(* IEC 61131-3 sources: std_i2980_v2.06_cp053/Source/IMM/ieccontrol/OutputCoordination1 (part 2) *)

(* ---- ABCoordList.pu ---- *)
IMPORT_OVER_LISTFILE
 SET_ALARM
, tsListStructCoord
, tsDeviceId
, FBDebugTrace
, tsTraceLevel
, tsElementCoord
, tsSearchDataCoord

END_IMPORT

ALGORITHM_BLOCK ABCoordList #DUMMY_EDIT_BLOCK

SYSTEM_VAR
 sv_DeviceId : tsDeviceId;
 sv_TraceLevel : tsTraceLevel;
END_VAR

SYSTEM_OBJECT
 erListOverflow : ALARM;
END_OBJECT

VAR
 mListStruct : tsListStructCoord;
 miNextFree : DINT;
 miLowBound : DINT;
 miHighBound : DINT;
 mbInit : BOOL;
 miLastFound : DINT;
 miActElement : DINT;
 fbDebugTrace : FBDebugTrace;
END_VAR

ALGORITHM aInit

#BEGIN_EDIT_BLOCK
miLowBound := GET_LOW_BOUND(mListStruct.List);
miHighBound := GET_HIGH_BOUND(mListStruct.List);
miNextFree := miLowBound;
miLastFound := miLowBound;
miActElement := miLowBound;
mbInit := TRUE;

;#END_EDIT_BLOCK END_ALGORITHM

ALGORITHM aAdd

VAR_INPUT
 Element : tsElementCoord;
END_VAR
#BEGIN_EDIT_BLOCK
IF NOT mbInit THEN RETURN;; END_IF;

IF miNextFree < miHighBound THEN

    mListStruct.List[miNextFree] := Element;
    mListStruct.Used[miNextFree] := TRUE;
    miNextFree := miNextFree + 1;
ELSE
    //error: List Full
    SET_ALARM(Name := erListOverflow,
              SubID1 := sv_DeviceId.CompId,
              SubID2 := sv_DeviceId.IndexId,
              Param1 := 'ABCoordList.aAdd');
END_IF;

;#END_EDIT_BLOCK END_ALGORITHM

ALGORITHM aAddAt

VAR_INPUT
 Element : tsElementCoord;
 iPos : DINT;
END_VAR

VAR_TEMP
 i : DINT;
END_VAR

VAR
 iStart : DINT;
 iEnd : DINT;
END_VAR
#BEGIN_EDIT_BLOCK
IF NOT mbInit THEN RETURN; END_IF;

IF miNextFree <= miHighBound THEN
    IF iPos < miHighBound AND iPos >= miLowBound THEN

        IF iPos < miNextFree THEN

            iStart := miNextFree;
            iEnd := iPos+1;
        ELSE
            i := iPos;
            iEnd := miNextFree;
        END_IF;
        miNextFree := i + 1;

        //reorganize list
        FOR i := iStart TO iEnd BY -1 DO
            mListStruct.List[i] := mListStruct.List[i-1];
            mListStruct.Used[i] := TRUE;
        END_FOR;
        //adding Element
        mListStruct.List[iPos] := Element;
        mListStruct.Used[iPos] := TRUE;
    ELSE
        //error: out of bounds
        IF sv_TraceLevel.bApplication THEN
            fbDebugTrace(sText := 'ABCoordList.aAddAt: Error: Out of ListBounds');
        END_IF;
    END_IF;
ELSE
    //error: List Full
    SET_ALARM(Name := erListOverflow,
            SubID1 := sv_DeviceId.CompId,
            SubID2 := sv_DeviceId.IndexId,
            Param1 := 'ABCoordList.aAddAt');
END_IF;

;#END_EDIT_BLOCK END_ALGORITHM

ALGORITHM aSearch

VAR_INPUT
 SearchData : tsSearchDataCoord;
END_VAR

VAR_OUTPUT
 Element : tsElementCoord;
 iPos : DINT;
 bFound : BOOL;
END_VAR

VAR_TEMP
 i : DINT;
END_VAR
#BEGIN_EDIT_BLOCK
IF NOT mbInit THEN RETURN; END_IF;

iPos := 0;
bFound := FALSE;

FOR i := miLowBound TO miNextFree-1 DO

    IF  mListStruct.Used[i] THEN
        IF mListStruct.List[i].SearchData = SearchData THEN

            Element := mListStruct.List[i];
            //remember foundposition for aSearchNext
            miLastFound := i;
            iPos := i;
            bFound := TRUE;
            RETURN;
        END_IF;
    ELSE
        EXIT;
    END_IF;
END_FOR;

;#END_EDIT_BLOCK END_ALGORITHM

ALGORITHM aSearchNext

VAR_INPUT
 SearchData : tsSearchDataCoord;
END_VAR

VAR_OUTPUT
 Element : tsElementCoord;
 iPos : DINT;
 bFound : BOOL;
END_VAR

VAR_TEMP
 i : DINT;
END_VAR
#BEGIN_EDIT_BLOCK
IF NOT mbInit THEN RETURN;; END_IF;

iPos := 0;
bFound := FALSE;

FOR i := miLastFound+1 TO miNextFree-1 DO

    IF mListStruct.List[i].SearchData = SearchData THEN

       Element := mListStruct.List[i];
       //remember foundposition for then next aSearchNext
       miLastFound := i;
       iPos := i;
       bFound := TRUE;
       RETURN;;
    END_IF;
END_FOR;

;#END_EDIT_BLOCK END_ALGORITHM

ALGORITHM aRemove

VAR_INPUT
 SearchData : tsSearchDataCoord;
END_VAR

VAR_OUTPUT
 Element : tsElementCoord;
 iPos : DINT;
 bFound : BOOL;
END_VAR

VAR_TEMP
 i : DINT;
END_VAR
#BEGIN_EDIT_BLOCK
IF NOT mbInit THEN RETURN; END_IF;

iPos := 0;
bFound := FALSE;

FOR i := miLowBound TO miNextFree-1 DO

    IF mListStruct.List[i].SearchData = SearchData AND mListStruct.Used[i] THEN

       iPos := i;
       bFound := TRUE;
       Element := mListStruct.List[i];
       //reorganize list
       FOR i := iPos TO miNextFree-1 DO
           mListStruct.List[i] := mListStruct.List[i+1];
       END_FOR;
       mListStruct.Used[miNextFree-1] := FALSE;
       miNextFree := miNextFree - 1;
       RETURN;
    END_IF;
END_FOR;

;#END_EDIT_BLOCK END_ALGORITHM

ALGORITHM aRemoveAt

VAR_INPUT
 iPos : DINT;
END_VAR

VAR_OUTPUT
 Element : tsElementCoord;
END_VAR

VAR_TEMP
 i : DINT;
END_VAR
#BEGIN_EDIT_BLOCK
IF NOT mbInit THEN RETURN; END_IF;

IF iPos <= miHighBound AND iPos >= miLowBound THEN

    Element:= mListStruct.List[iPos];
    miActElement := iPos;

    //reorganize list
    FOR i := iPos TO miNextFree-1 DO
        mListStruct.List[i] := mListStruct.List[i+1];
        mListStruct.Used[i] := mListStruct.Used[i+1];
    END_FOR;
    mListStruct.Used[miNextFree-1] := FALSE;

    miNextFree := miNextFree - 1;
ELSE
    //error: out of bounds
    IF sv_TraceLevel.bApplication THEN
        fbDebugTrace(sText := 'ABCoordList.aRemoveAt: Error: Out of ListBounds');
    END_IF;
END_IF;

;#END_EDIT_BLOCK END_ALGORITHM

ALGORITHM aRemoveAll

VAR_TEMP
 i : DINT;
END_VAR
#BEGIN_EDIT_BLOCK
IF NOT mbInit THEN RETURN; END_IF;
FOR i := miNextFree-1 TO miLowBound DO
    //clearing the whole list
    mListStruct.Used[i] := FALSE;
END_FOR;
miNextFree := miLowBound;

;#END_EDIT_BLOCK END_ALGORITHM

ALGORITHM aElementAt

VAR_OUTPUT
 Element : tsElementCoord;
END_VAR

VAR_INPUT
 iPos : DINT;
END_VAR
#BEGIN_EDIT_BLOCK
IF NOT mbInit THEN RETURN; END_IF;

IF iPos <= miHighBound AND iPos >= miLowBound THEN

    Element := mListStruct.List[iPos];
    miActElement := iPos;
ELSE
    //error: out of bounds
    IF sv_TraceLevel.bApplication THEN
        fbDebugTrace(sText := 'ABCoordList.aElementAt: Error: Out of ListBounds');
    END_IF;
END_IF;

;#END_EDIT_BLOCK END_ALGORITHM

ALGORITHM aModifyAt

VAR_INPUT
 iPos : DINT;
 Element : tsElementCoord;
END_VAR
#BEGIN_EDIT_BLOCK
IF NOT mbInit THEN RETURN; END_IF;

IF iPos <= miHighBound AND iPos >= miLowBound THEN

     mListStruct.List[iPos] := Element;
     miActElement := iPos;
ELSE
    //error: out of bounds
    IF sv_TraceLevel.bApplication THEN
        fbDebugTrace(sText := 'ABCoordList.aModifyAt: Error: Out of ListBounds');
    END_IF;
END_IF;

;#END_EDIT_BLOCK END_ALGORITHM

FUNCTION aGetSize : DINT
 #DUMMY_EDIT_BLOCK
#BEGIN_EDIT_BLOCK
IF NOT mbInit THEN RETURN; END_IF;
//returns the size of the list
aGetSize := miHighBound - miLowBound;

;#END_EDIT_BLOCK END_FUNCTION

FUNCTION aGetElementCount : DINT
 #DUMMY_EDIT_BLOCK
#BEGIN_EDIT_BLOCK
IF NOT mbInit THEN RETURN; END_IF;

aGetElementCount:= miNextFree - miLowBound;

;#END_EDIT_BLOCK END_FUNCTION

ALGORITHM aFirstElement

VAR_OUTPUT
 Element : tsElementCoord;
END_VAR
#BEGIN_EDIT_BLOCK
IF NOT mbInit THEN RETURN; END_IF;

miActElement := miLowBound;
Element := mListStruct.List[miLowBound];

;#END_EDIT_BLOCK END_ALGORITHM

ALGORITHM aNextElement

VAR_OUTPUT
 Element : tsElementCoord;
 iPos : DINT;
END_VAR
#BEGIN_EDIT_BLOCK
IF NOT mbInit THEN RETURN; END_IF;

IF miActElement < miHighBound THEN

    miActElement := miActElement + 1;
    iPos := miActElement;
    Element := mListStruct.List[miActElement];
END_IF;

;#END_EDIT_BLOCK END_ALGORITHM

ALGORITHM aLastElement

VAR_OUTPUT
 Element : tsElementCoord;
END_VAR
#BEGIN_EDIT_BLOCK
IF NOT mbInit THEN RETURN; END_IF;

miActElement := miNextFree - 1;
Element := mListStruct.List[miActElement];

;#END_EDIT_BLOCK END_ALGORITHM

ALGORITHM aPrevElement

VAR_OUTPUT
 Element : tsElementCoord;
 iPos : DINT;
END_VAR
#BEGIN_EDIT_BLOCK
IF NOT mbInit THEN RETURN; END_IF;

IF miActElement > miLowBound THEN

    miActElement := miActElement - 1;
    iPos := miActElement;
    Element := mListStruct.List[miActElement];
END_IF;

;#END_EDIT_BLOCK END_ALGORITHM

ALGORITHM aImport

VAR_INPUT
 ListStruct : tsListStructCoord;
END_VAR

VAR_TEMP
 i : DINT;
END_VAR
#BEGIN_EDIT_BLOCK
IF NOT mbInit THEN RETURN; END_IF;

miLastFound := miLowBound;
miActElement := miLowBound;
miNextFree := miLowBound;
mListStruct :=  ListStruct;

//cheching used elements
FOR i := miLowBound TO miHighBound DO

   IF NOT mListStruct.Used[i] THEN
        miNextFree := i;
        RETURN;
   END_IF;
END_FOR;

;#END_EDIT_BLOCK END_ALGORITHM

ALGORITHM aExport

VAR_OUTPUT
 ListStruct : tsListStructCoord;
END_VAR
#BEGIN_EDIT_BLOCK
IF NOT mbInit THEN RETURN; END_IF;

ListStruct := mListStruct;

;#END_EDIT_BLOCK END_ALGORITHM

END_ALGORITHM_BLOCK

#END_OF_IEC_PART

@Puma @IecEditor 6 68 @Pou 25
@@@BEG_Comment@@@

@@@END_Comment@@@

@BEG_Contents

@BEG_Func
@RT(17)FuncTreeContainer
1
@Var @RT(9)SET_ALARM @RT(0) @T @T @DERIVED 0 @F @RT(23)KEBA_STANDARD_PROCEDURE @F
@T
@BEG_Attrib
0 @RT(0) @RT(0)
@END_Attrib
1 1 @F @F @F @F

@END_Func

@BEG_Const
@RT(18)ConstTreeContainer
0
@END_Const

@BEG_Export

@BEG_Kind
@ALGORITHM_BLOCK @RT(11)ABCoordList @STRUCTURED_TEXT
@RT(0) @RT(0) @RT(0)
@END_Kind

@BEG_Dcl
@RT(16)DclTreeContainer
11
@Var @RT(14)erListOverflow @RT(0) @T @F @DT @RT(5)ALARM @RT(0) @T @T @BASIC 0 @F
@F @F
@T
@BEG_Attrib
3 @RT(0) @RT(0) @RT(0)
@END_Attrib
1 7 @F @F @F @F

@Var @RT(11)mListStruct @RT(0) @T @T @DERIVED 0 @T @T @DT @RT(17)tsListStructCoord @RT(0) @T @T @UNKNOWN 0 @F
@F @F
@T
@BEG_Attrib
3 @RT(0) @RT(0) @RT(0)
@END_Attrib
1 0 @F @F @F @F

@Var @RT(10)miNextFree @RT(0) @T @F @DT @RT(4)DINT @RT(0) @T @T @BASIC 0 @F
@F @F
@T
@BEG_Attrib
3 @RT(0) @RT(0) @RT(0)
@END_Attrib
1 0 @F @F @F @F

@Var @RT(10)miLowBound @RT(0) @T @F @DT @RT(4)DINT @RT(0) @T @T @BASIC 0 @F
@F @F
@T
@BEG_Attrib
3 @RT(0) @RT(0) @RT(0)
@END_Attrib
1 0 @F @F @F @F

@Var @RT(11)miHighBound @RT(0) @T @F @DT @RT(4)DINT @RT(0) @T @T @BASIC 0 @F
@F @F
@T
@BEG_Attrib
3 @RT(0) @RT(0) @RT(0)
@END_Attrib
1 0 @F @F @F @F

@Var @RT(6)mbInit @RT(0) @T @F @DT @RT(4)BOOL @RT(0) @T @T @BASIC 0 @F
@F @F
@T
@BEG_Attrib
3 @RT(0) @RT(0) @RT(0)
@END_Attrib
1 0 @F @F @F @F

@Var @RT(11)miLastFound @RT(0) @T @F @DT @RT(4)DINT @RT(0) @T @T @BASIC 0 @F
@F @F
@T
@BEG_Attrib
3 @RT(0) @RT(0) @RT(0)
@END_Attrib
1 0 @F @F @F @F

@Var @RT(12)miActElement @RT(0) @T @F @DT @RT(4)DINT @RT(0) @T @T @BASIC 0 @F
@F @F
@T
@BEG_Attrib
3 @RT(0) @RT(0) @RT(0)
@END_Attrib
1 0 @F @F @F @F

@Var @RT(11)sv_DeviceId @RT(0) @T @T @DERIVED 0 @T @T @DT @RT(10)tsDeviceId @RT(0) @T @T @UNKNOWN 0 @F
@F @F
@T
@BEG_Attrib
3 @RT(0) @RT(0) @RT(0)
@END_Attrib
1 8 @F @F @F @F

@Var @RT(12)fbDebugTrace @RT(0) @T @T @DERIVED 0 @T @T @DT @RT(12)FBDebugTrace @RT(0) @T @T @UNKNOWN 0 @F
@F @F
@T
@BEG_Attrib
3 @RT(0) @RT(0) @RT(0)
@END_Attrib
1 0 @F @F @F @F

@Var @RT(13)sv_TraceLevel @RT(0) @T @T @DERIVED 0 @T @T @DT @RT(12)tsTraceLevel @RT(0) @T @T @UNKNOWN 0 @F
@F @F
@T
@BEG_Attrib
3 @RT(0) @RT(0) @RT(0)
@END_Attrib
1 8 @F @F @F @F

@END_Dcl

@END_Export

@BEG_Body

18

@BEG_Export

@BEG_Algo
@ALGORITHM @RT(5)aInit @STRUCTURED_TEXT
@RT(0) @RT(0) @RT(0) @F @F
@END_Algo

@BEG_Dcl
@RT(16)DclTreeContainer
0
@END_Dcl

@END_Export

@BEG_Export

@BEG_Algo
@ALGORITHM @RT(4)aAdd @STRUCTURED_TEXT
@RT(0) @RT(0) @RT(0) @F @F
@END_Algo

@BEG_Dcl
@RT(16)DclTreeContainer
1
@Var @RT(7)Element @RT(0) @T @T @DERIVED 0 @T @T @DT @RT(14)tsElementCoord @RT(0) @T @T @UNKNOWN 0 @F
@F @F
@T
@BEG_Attrib
3 @RT(0) @RT(0) @RT(0)
@END_Attrib
1 1 @F @F @F @F

@END_Dcl

@END_Export

@BEG_Export

@BEG_Algo
@ALGORITHM @RT(6)aAddAt @STRUCTURED_TEXT
@RT(0) @RT(0) @RT(0) @F @F
@END_Algo

@BEG_Dcl
@RT(16)DclTreeContainer
5
@Var @RT(7)Element @RT(0) @T @T @DERIVED 0 @T @T @DT @RT(14)tsElementCoord @RT(0) @T @T @UNKNOWN 0 @F
@F @F
@T
@BEG_Attrib
3 @RT(0) @RT(0) @RT(0)
@END_Attrib
1 1 @F @F @F @F

@Var @RT(4)iPos @RT(0) @T @F @DT @RT(4)DINT @RT(0) @T @T @BASIC 0 @F
@F @F
@T
@BEG_Attrib
3 @RT(0) @RT(0) @RT(0)
@END_Attrib
1 1 @F @F @F @F

@Var @RT(1)i @RT(0) @T @F @DT @RT(4)DINT @RT(0) @T @T @BASIC 0 @F
@F @F
@T
@BEG_Attrib
3 @RT(0) @RT(0) @RT(0)
@END_Attrib
1 4 @F @F @F @F

@Var @RT(6)iStart @RT(0) @T @F @DT @RT(4)DINT @RT(0) @T @T @BASIC 0 @F
@F @F
@T
@BEG_Attrib
3 @RT(0) @RT(0) @RT(0)
@END_Attrib
1 0 @F @F @F @F

@Var @RT(4)iEnd @RT(0) @T @F @DT @RT(4)DINT @RT(0) @T @T @BASIC 0 @F
@F @F
@T
@BEG_Attrib
3 @RT(0) @RT(0) @RT(0)
@END_Attrib
1 0 @F @F @F @F

@END_Dcl

@END_Export

@BEG_Export

@BEG_Algo
@ALGORITHM @RT(7)aSearch @STRUCTURED_TEXT
@RT(0) @RT(0) @RT(0) @F @F
@END_Algo

@BEG_Dcl
@RT(16)DclTreeContainer
5
@Var @RT(10)SearchData @RT(0) @T @T @DERIVED 0 @T @T @DT @RT(17)tsSearchDataCoord @RT(0) @T @T @UNKNOWN 0 @F
@F @F
@T
@BEG_Attrib
3 @RT(0) @RT(0) @RT(0)
@END_Attrib
1 1 @F @F @F @F

@Var @RT(7)Element @RT(0) @T @T @DERIVED 0 @T @T @DT @RT(14)tsElementCoord @RT(0) @T @T @UNKNOWN 0 @F
@F @F
@T
@BEG_Attrib
3 @RT(0) @RT(0) @RT(0)
@END_Attrib
1 3 @F @F @F @F

@Var @RT(4)iPos @RT(0) @T @F @DT @RT(4)DINT @RT(0) @T @T @BASIC 0 @F
@F @F
@T
@BEG_Attrib
3 @RT(0) @RT(0) @RT(0)
@END_Attrib
1 3 @F @F @F @F

@Var @RT(6)bFound @RT(0) @T @F @DT @RT(4)BOOL @RT(0) @T @T @BASIC 0 @F
@F @F
@T
@BEG_Attrib
3 @RT(0) @RT(0) @RT(0)
@END_Attrib
1 3 @F @F @F @F

@Var @RT(1)i @RT(0) @T @F @DT @RT(4)DINT @RT(0) @T @T @BASIC 0 @F
@F @F
@T
@BEG_Attrib
3 @RT(0) @RT(0) @RT(0)
@END_Attrib
1 4 @F @F @F @F

@END_Dcl

@END_Export

@BEG_Export

@BEG_Algo
@ALGORITHM @RT(11)aSearchNext @STRUCTURED_TEXT
@RT(0) @RT(0) @RT(0) @F @F
@END_Algo

@BEG_Dcl
@RT(16)DclTreeContainer
5
@Var @RT(10)SearchData @RT(0) @T @T @DERIVED 0 @T @T @DT @RT(17)tsSearchDataCoord @RT(0) @T @T @UNKNOWN 0 @F
@F @F
@T
@BEG_Attrib
3 @RT(0) @RT(0) @RT(0)
@END_Attrib
1 1 @F @F @F @F

@Var @RT(7)Element @RT(0) @T @T @DERIVED 0 @T @T @DT @RT(14)tsElementCoord @RT(0) @T @T @UNKNOWN 0 @F
@F @F
@T
@BEG_Attrib
3 @RT(0) @RT(0) @RT(0)
@END_Attrib
1 3 @F @F @F @F

@Var @RT(4)iPos @RT(0) @T @F @DT @RT(4)DINT @RT(0) @T @T @BASIC 0 @F
@F @F
@T
@BEG_Attrib
3 @RT(0) @RT(0) @RT(0)
@END_Attrib
1 3 @F @F @F @F

@Var @RT(6)bFound @RT(0) @T @F @DT @RT(4)BOOL @RT(0) @T @T @BASIC 0 @F
@F @F
@T
@BEG_Attrib
3 @RT(0) @RT(0) @RT(0)
@END_Attrib
1 3 @F @F @F @F

@Var @RT(1)i @RT(0) @T @F @DT @RT(4)DINT @RT(0) @T @T @BASIC 0 @F
@F @F
@T
@BEG_Attrib
3 @RT(0) @RT(0) @RT(0)
@END_Attrib
1 4 @F @F @F @F

@END_Dcl

@END_Export

@BEG_Export

@BEG_Algo
@ALGORITHM @RT(7)aRemove @STRUCTURED_TEXT
@RT(0) @RT(0) @RT(0) @F @F
@END_Algo

@BEG_Dcl
@RT(16)DclTreeContainer
5
@Var @RT(10)SearchData @RT(0) @T @T @DERIVED 0 @T @T @DT @RT(17)tsSearchDataCoord @RT(0) @T @T @UNKNOWN 0 @F
@F @F
@T
@BEG_Attrib
3 @RT(0) @RT(0) @RT(0)
@END_Attrib
1 1 @F @F @F @F

@Var @RT(7)Element @RT(0) @T @T @DERIVED 0 @T @T @DT @RT(14)tsElementCoord @RT(0) @T @T @UNKNOWN 0 @F
@F @F
@T
@BEG_Attrib
3 @RT(0) @RT(0) @RT(0)
@END_Attrib
1 3 @F @F @F @F

@Var @RT(4)iPos @RT(0) @T @F @DT @RT(4)DINT @RT(0) @T @T @BASIC 0 @F
@F @F
@T
@BEG_Attrib
3 @RT(0) @RT(0) @RT(0)
@END_Attrib
1 3 @F @F @F @F

@Var @RT(6)bFound @RT(0) @T @F @DT @RT(4)BOOL @RT(0) @T @T @BASIC 0 @F
@F @F
@T
@BEG_Attrib
3 @RT(0) @RT(0) @RT(0)
@END_Attrib
1 3 @F @F @F @F

@Var @RT(1)i @RT(0) @T @F @DT @RT(4)DINT @RT(0) @T @T @BASIC 0 @F
@F @F
@T
@BEG_Attrib
3 @RT(0) @RT(0) @RT(0)
@END_Attrib
1 4 @F @F @F @F

@END_Dcl

@END_Export

@BEG_Export

@BEG_Algo
@ALGORITHM @RT(9)aRemoveAt @STRUCTURED_TEXT
@RT(0) @RT(0) @RT(0) @F @F
@END_Algo

@BEG_Dcl
@RT(16)DclTreeContainer
3
@Var @RT(4)iPos @RT(0) @T @F @DT @RT(4)DINT @RT(0) @T @T @BASIC 0 @F
@F @F
@T
@BEG_Attrib
3 @RT(0) @RT(0) @RT(0)
@END_Attrib
1 1 @F @F @F @F

@Var @RT(7)Element @RT(0) @T @T @DERIVED 0 @T @T @DT @RT(14)tsElementCoord @RT(0) @T @T @UNKNOWN 0 @F
@F @F
@T
@BEG_Attrib
3 @RT(0) @RT(0) @RT(0)
@END_Attrib
1 3 @F @F @F @F

@Var @RT(1)i @RT(0) @T @F @DT @RT(4)DINT @RT(0) @T @T @BASIC 0 @F
@F @F
@T
@BEG_Attrib
3 @RT(0) @RT(0) @RT(0)
@END_Attrib
1 4 @F @F @F @F

@END_Dcl

@END_Export

@BEG_Export

@BEG_Algo
@ALGORITHM @RT(10)aRemoveAll @STRUCTURED_TEXT
@RT(0) @RT(0) @RT(0) @F @F
@END_Algo

@BEG_Dcl
@RT(16)DclTreeContainer
1
@Var @RT(1)i @RT(0) @T @F @DT @RT(4)DINT @RT(0) @T @T @BASIC 0 @F
@F @F
@T
@BEG_Attrib
3 @RT(0) @RT(0) @RT(0)
@END_Attrib
1 4 @F @F @F @F

@END_Dcl

@END_Export

@BEG_Export

@BEG_Algo
@ALGORITHM @RT(10)aElementAt @STRUCTURED_TEXT
@RT(0) @RT(0) @RT(0) @F @F
@END_Algo

@BEG_Dcl
@RT(16)DclTreeContainer
2
@Var @RT(7)Element @RT(0) @T @T @DERIVED 0 @T @T @DT @RT(14)tsElementCoord @RT(0) @T @T @UNKNOWN 0 @F
@F @F
@T
@BEG_Attrib
3 @RT(0) @RT(0) @RT(0)
@END_Attrib
1 3 @F @F @F @F

@Var @RT(4)iPos @RT(0) @T @F @DT @RT(4)DINT @RT(0) @T @T @BASIC 0 @F
@F @F
@T
@BEG_Attrib
3 @RT(0) @RT(0) @RT(0)
@END_Attrib
1 1 @F @F @F @F

@END_Dcl

@END_Export

@BEG_Export

@BEG_Algo
@ALGORITHM @RT(9)aModifyAt @STRUCTURED_TEXT
@RT(0) @RT(0) @RT(0) @F @F
@END_Algo

@BEG_Dcl
@RT(16)DclTreeContainer
2
@Var @RT(4)iPos @RT(0) @T @F @DT @RT(4)DINT @RT(0) @T @T @BASIC 0 @F
@F @F
@T
@BEG_Attrib
3 @RT(0) @RT(0) @RT(0)
@END_Attrib
1 1 @F @F @F @F

@Var @RT(7)Element @RT(0) @T @T @DERIVED 0 @T @T @DT @RT(14)tsElementCoord @RT(0) @T @T @UNKNOWN 0 @F
@F @F
@T
@BEG_Attrib
3 @RT(0) @RT(0) @RT(0)
@END_Attrib
1 1 @F @F @F @F

@END_Dcl

@END_Export

@BEG_Export

@BEG_Algo
@FUNCTION @RT(8)aGetSize @STRUCTURED_TEXT
@RT(4)DINT @RT(0) @RT(0) @F @F
@END_Algo

@BEG_Dcl
@RT(16)DclTreeContainer
0
@END_Dcl

@END_Export

@BEG_Export

@BEG_Algo
@FUNCTION @RT(16)aGetElementCount @STRUCTURED_TEXT
@RT(4)DINT @RT(0) @RT(0) @F @F
@END_Algo

@BEG_Dcl
@RT(16)DclTreeContainer
0
@END_Dcl

@END_Export

@BEG_Export

@BEG_Algo
@ALGORITHM @RT(13)aFirstElement @STRUCTURED_TEXT
@RT(0) @RT(0) @RT(0) @F @F
@END_Algo

@BEG_Dcl
@RT(16)DclTreeContainer
1
@Var @RT(7)Element @RT(0) @T @T @DERIVED 0 @T @T @DT @RT(14)tsElementCoord @RT(0) @T @T @UNKNOWN 0 @F
@F @F
@T
@BEG_Attrib
3 @RT(0) @RT(0) @RT(0)
@END_Attrib
1 3 @F @F @F @F

@END_Dcl

@END_Export

@BEG_Export

@BEG_Algo
@ALGORITHM @RT(12)aNextElement @STRUCTURED_TEXT
@RT(0) @RT(0) @RT(0) @F @F
@END_Algo

@BEG_Dcl
@RT(16)DclTreeContainer
2
@Var @RT(7)Element @RT(0) @T @T @DERIVED 0 @T @T @DT @RT(14)tsElementCoord @RT(0) @T @T @UNKNOWN 0 @F
@F @F
@T
@BEG_Attrib
3 @RT(0) @RT(0) @RT(0)
@END_Attrib
1 3 @F @F @F @F

@Var @RT(4)iPos @RT(0) @T @F @DT @RT(4)DINT @RT(0) @T @T @BASIC 0 @F
@F @F
@T
@BEG_Attrib
3 @RT(0) @RT(0) @RT(0)
@END_Attrib
1 3 @F @F @F @F

@END_Dcl

@END_Export

@BEG_Export

@BEG_Algo
@ALGORITHM @RT(12)aLastElement @STRUCTURED_TEXT
@RT(0) @RT(0) @RT(0) @F @F
@END_Algo

@BEG_Dcl
@RT(16)DclTreeContainer
1
@Var @RT(7)Element @RT(0) @T @T @DERIVED 0 @T @T @DT @RT(14)tsElementCoord @RT(0) @T @T @UNKNOWN 0 @F
@F @F
@T
@BEG_Attrib
3 @RT(0) @RT(0) @RT(0)
@END_Attrib
1 3 @F @F @F @F

@END_Dcl

@END_Export

@BEG_Export

@BEG_Algo
@ALGORITHM @RT(12)aPrevElement @STRUCTURED_TEXT
@RT(0) @RT(0) @RT(0) @F @F
@END_Algo

@BEG_Dcl
@RT(16)DclTreeContainer
2
@Var @RT(7)Element @RT(0) @T @T @DERIVED 0 @T @T @DT @RT(14)tsElementCoord @RT(0) @T @T @UNKNOWN 0 @F
@F @F
@T
@BEG_Attrib
3 @RT(0) @RT(0) @RT(0)
@END_Attrib
1 3 @F @F @F @F

@Var @RT(4)iPos @RT(0) @T @F @DT @RT(4)DINT @RT(0) @T @T @BASIC 0 @F
@F @F
@T
@BEG_Attrib
3 @RT(0) @RT(0) @RT(0)
@END_Attrib
1 3 @F @F @F @F

@END_Dcl

@END_Export

@BEG_Export

@BEG_Algo
@ALGORITHM @RT(7)aImport @STRUCTURED_TEXT
@RT(0) @RT(0) @RT(0) @F @F
@END_Algo

@BEG_Dcl
@RT(16)DclTreeContainer
2
@Var @RT(10)ListStruct @RT(0) @T @T @DERIVED 0 @T @T @DT @RT(17)tsListStructCoord @RT(0) @T @T @UNKNOWN 0 @F
@F @F
@T
@BEG_Attrib
3 @RT(0) @RT(0) @RT(0)
@END_Attrib
1 1 @F @F @F @F

@Var @RT(1)i @RT(0) @T @F @DT @RT(4)DINT @RT(0) @T @T @BASIC 0 @F
@F @F
@T
@BEG_Attrib
3 @RT(0) @RT(0) @RT(0)
@END_Attrib
1 4 @F @F @F @F

@END_Dcl

@END_Export

@BEG_Export

@BEG_Algo
@ALGORITHM @RT(7)aExport @STRUCTURED_TEXT
@RT(0) @RT(0) @RT(0) @F @F
@END_Algo

@BEG_Dcl
@RT(16)DclTreeContainer
1
@Var @RT(10)ListStruct @RT(0) @T @T @DERIVED 0 @T @T @DT @RT(17)tsListStructCoord @RT(0) @T @T @UNKNOWN 0 @F
@F @F
@T
@BEG_Attrib
3 @RT(0) @RT(0) @RT(0)
@END_Attrib
1 3 @F @F @F @F

@END_Dcl

@END_Export

@BEG_Body
@TL(7)
miLowBound := GET_LOW_BOUND(mListStruct.List);
miHighBound := GET_HIGH_BOUND(mListStruct.List);
miNextFree := miLowBound;
miLastFound := miLowBound;
miActElement := miLowBound;
mbInit := TRUE;

@END_Body

@@@BEG_Comment@@@
@TL(0)

@@@END_Comment@@@

@BEG_Body
@TL(15)
IF NOT mbInit THEN RETURN;; END_IF;

IF miNextFree < miHighBound THEN

    mListStruct.List[miNextFree] := Element;
    mListStruct.Used[miNextFree] := TRUE;
    miNextFree := miNextFree + 1;
ELSE
    //error: List Full
    SET_ALARM(Name := erListOverflow,
              SubID1 := sv_DeviceId.CompId,
              SubID2 := sv_DeviceId.IndexId,
              Param1 := 'ABCoordList.aAdd');
END_IF;

@END_Body

@@@BEG_Comment@@@
@TL(0)

@@@END_Comment@@@

@BEG_Body
@TL(37)
IF NOT mbInit THEN RETURN; END_IF;

IF miNextFree <= miHighBound THEN
    IF iPos < miHighBound AND iPos >= miLowBound THEN

        IF iPos < miNextFree THEN

            iStart := miNextFree;
            iEnd := iPos+1;
        ELSE
            i := iPos;
            iEnd := miNextFree;
        END_IF;
        miNextFree := i + 1;

        //reorganize list
        FOR i := iStart TO iEnd BY -1 DO
            mListStruct.List[i] := mListStruct.List[i-1];
            mListStruct.Used[i] := TRUE;
        END_FOR;
        //adding Element
        mListStruct.List[iPos] := Element;
        mListStruct.Used[iPos] := TRUE;
    ELSE
        //error: out of bounds
        IF sv_TraceLevel.bApplication THEN
            fbDebugTrace(sText := 'ABCoordList.aAddAt: Error: Out of ListBounds');
        END_IF;
    END_IF;
ELSE
    //error: List Full
    SET_ALARM(Name := erListOverflow,
            SubID1 := sv_DeviceId.CompId,
            SubID2 := sv_DeviceId.IndexId,
            Param1 := 'ABCoordList.aAddAt');
END_IF;

@END_Body

@@@BEG_Comment@@@
@TL(0)

@@@END_Comment@@@

@BEG_Body
@TL(22)
IF NOT mbInit THEN RETURN; END_IF;

iPos := 0;
bFound := FALSE;

FOR i := miLowBound TO miNextFree-1 DO

    IF  mListStruct.Used[i] THEN
        IF mListStruct.List[i].SearchData = SearchData THEN

            Element := mListStruct.List[i];
            //remember foundposition for aSearchNext
            miLastFound := i;
            iPos := i;
            bFound := TRUE;
            RETURN;
        END_IF;
    ELSE
        EXIT;
    END_IF;
END_FOR;

@END_Body

@@@BEG_Comment@@@
@TL(0)

@@@END_Comment@@@

@BEG_Body
@TL(19)
IF NOT mbInit THEN RETURN;; END_IF;

iPos := 0;
bFound := FALSE;

FOR i := miLastFound+1 TO miNextFree-1 DO

    IF mListStruct.List[i].SearchData = SearchData THEN

       Element := mListStruct.List[i];
       //remember foundposition for then next aSearchNext
       miLastFound := i;
       iPos := i;
       bFound := TRUE;
       RETURN;;
    END_IF;
END_FOR;

@END_Body

@@@BEG_Comment@@@
@TL(0)

@@@END_Comment@@@

@BEG_Body
@TL(22)
IF NOT mbInit THEN RETURN; END_IF;

iPos := 0;
bFound := FALSE;

FOR i := miLowBound TO miNextFree-1 DO

    IF mListStruct.List[i].SearchData = SearchData AND mListStruct.Used[i] THEN

       iPos := i;
       bFound := TRUE;
       Element := mListStruct.List[i];
       //reorganize list
       FOR i := iPos TO miNextFree-1 DO
           mListStruct.List[i] := mListStruct.List[i+1];
       END_FOR;
       mListStruct.Used[miNextFree-1] := FALSE;
       miNextFree := miNextFree - 1;
       RETURN;
    END_IF;
END_FOR;

@END_Body

@@@BEG_Comment@@@
@TL(0)

@@@END_Comment@@@

@BEG_Body
@TL(22)
IF NOT mbInit THEN RETURN; END_IF;

IF iPos <= miHighBound AND iPos >= miLowBound THEN

    Element:= mListStruct.List[iPos];
    miActElement := iPos;

    //reorganize list
    FOR i := iPos TO miNextFree-1 DO
        mListStruct.List[i] := mListStruct.List[i+1];
        mListStruct.Used[i] := mListStruct.Used[i+1];
    END_FOR;
    mListStruct.Used[miNextFree-1] := FALSE;

    miNextFree := miNextFree - 1;
ELSE
    //error: out of bounds
    IF sv_TraceLevel.bApplication THEN
        fbDebugTrace(sText := 'ABCoordList.aRemoveAt: Error: Out of ListBounds');
    END_IF;
END_IF;

@END_Body

@@@BEG_Comment@@@
@TL(0)

@@@END_Comment@@@

@BEG_Body
@TL(7)
IF NOT mbInit THEN RETURN; END_IF;
FOR i := miNextFree-1 TO miLowBound DO
    //clearing the whole list
    mListStruct.Used[i] := FALSE;
END_FOR;
miNextFree := miLowBound;

@END_Body

@@@BEG_Comment@@@
@TL(0)

@@@END_Comment@@@

@BEG_Body
@TL(13)
IF NOT mbInit THEN RETURN; END_IF;

IF iPos <= miHighBound AND iPos >= miLowBound THEN

    Element := mListStruct.List[iPos];
    miActElement := iPos;
ELSE
    //error: out of bounds
    IF sv_TraceLevel.bApplication THEN
        fbDebugTrace(sText := 'ABCoordList.aElementAt: Error: Out of ListBounds');
    END_IF;
END_IF;

@END_Body

@@@BEG_Comment@@@
@TL(0)

@@@END_Comment@@@

@BEG_Body
@TL(13)
IF NOT mbInit THEN RETURN; END_IF;

IF iPos <= miHighBound AND iPos >= miLowBound THEN

     mListStruct.List[iPos] := Element;
     miActElement := iPos;
ELSE
    //error: out of bounds
    IF sv_TraceLevel.bApplication THEN
        fbDebugTrace(sText := 'ABCoordList.aModifyAt: Error: Out of ListBounds');
    END_IF;
END_IF;

@END_Body

@@@BEG_Comment@@@
@TL(0)

@@@END_Comment@@@

@BEG_Body
@TL(5)
IF NOT mbInit THEN RETURN; END_IF;
//returns the size of the list
aGetSize := miHighBound - miLowBound;

@END_Body

@@@BEG_Comment@@@
@TL(0)

@@@END_Comment@@@

@BEG_Body
@TL(5)
IF NOT mbInit THEN RETURN; END_IF;

aGetElementCount:= miNextFree - miLowBound;

@END_Body

@@@BEG_Comment@@@
@TL(0)

@@@END_Comment@@@

@BEG_Body
@TL(6)
IF NOT mbInit THEN RETURN; END_IF;

miActElement := miLowBound;
Element := mListStruct.List[miLowBound];

@END_Body

@@@BEG_Comment@@@
@TL(0)

@@@END_Comment@@@

@BEG_Body
@TL(9)
IF NOT mbInit THEN RETURN; END_IF;

IF miActElement < miHighBound THEN

    miActElement := miActElement + 1;
    iPos := miActElement;
    Element := mListStruct.List[miActElement];
END_IF;

@END_Body

@@@BEG_Comment@@@
@TL(0)

@@@END_Comment@@@

@BEG_Body
@TL(6)
IF NOT mbInit THEN RETURN; END_IF;

miActElement := miNextFree - 1;
Element := mListStruct.List[miActElement];

@END_Body

@@@BEG_Comment@@@
@TL(0)

@@@END_Comment@@@

@BEG_Body
@TL(9)
IF NOT mbInit THEN RETURN; END_IF;

IF miActElement > miLowBound THEN

    miActElement := miActElement - 1;
    iPos := miActElement;
    Element := mListStruct.List[miActElement];
END_IF;

@END_Body

@@@BEG_Comment@@@
@TL(0)

@@@END_Comment@@@

@BEG_Body
@TL(16)
IF NOT mbInit THEN RETURN; END_IF;

miLastFound := miLowBound;
miActElement := miLowBound;
miNextFree := miLowBound;
mListStruct :=  ListStruct;

//cheching used elements
FOR i := miLowBound TO miHighBound DO

   IF NOT mListStruct.Used[i] THEN
        miNextFree := i;
        RETURN;
   END_IF;
END_FOR;

@END_Body

@@@BEG_Comment@@@
@TL(0)

@@@END_Comment@@@

@BEG_Body
@TL(4)
IF NOT mbInit THEN RETURN; END_IF;

ListStruct := mListStruct;

@END_Body

@@@BEG_Comment@@@
@TL(0)

@@@END_Comment@@@
@END_Body

@END_Contents

(* ---- ABPumpCombination.pu ---- *)
(*
@h    ! WARNING !
@h    The Kemro K2 system (including software) only meets category B according to EN 954-1,
@h    thus it is not intended for usage in safety-relevant control applications in the field
@h    of personal safety (e.g. emergency stop).
@h    To implement potentially necessary safety-relevant control tasks, always use additional
@h    external safety devices that are intended for the particular purpose, and meet the necessary
@h    functional safety.
@h    For further information see EN 954-1 (EN ISO 13849-1) and/or the K2-x00 user manual, chapter
@h    "CE conformity, directives and standards".

Algorithm block for setting hydraulic specific valves to link different pumps.
*)

IMPORT_OVER_LISTFILE
 tyPumpData

END_IMPORT

ALGORITHM_BLOCK ABPumpCombination #DUMMY_EDIT_BLOCK

SYSTEM_VAR
 do_LinkP1P2 : BOOL (* DO for linking Pump1 and Pump2 *);
 sv_PumpData : tyPumpData;
END_VAR

SYSTEM_OBJECT
 TaskInject : TASK;
 TaskMid : TASK;
END_OBJECT

PROCESS_ALGORITHM paInit ON TaskMid AUTOSTART

#BEGIN_EDIT_BLOCK
(**************************************** WARNING ********************************************
 *** The KEBA Kemro K2 System including software is not intended for safety control tasks! ***
 ***                       For further information see Comment tab!                        ***
 *********************************************************************************************)

IF IS_LINKED(do_LinkP1P2) THEN
   START_PROCESS_ALGORITHM(paLinkPump1Pump2);
END_IF;

STOP_PROCESS_ALGORITHM();

;#END_EDIT_BLOCK END_ALGORITHM

PROCESS_ALGORITHM paLinkPump1Pump2 ON TaskInject

VAR
 bSetDO : BOOL;
END_VAR

(* IecGraph-Code *)

(* init step *)
INITIAL_STEP S_Init:
END_STEP

(* steps *)
STEP S_Idle:
Action5 (N);
END_STEP

ACTION Action5: #BEGIN_EDIT_BLOCK
//set DO if a device actually outputs to both pumps
bSetDO := (sv_PumpData[1].PumpState = nPumpStateBusy) AND
          (sv_PumpData[2].PumpState = nPumpStateBusy) AND
          (sv_PumpData[1].ActiveDevice = sv_PumpData[2].ActiveDevice);

;#END_EDIT_BLOCK END_ACTION (*Action5*)
STEP S_Set_DO:
ASetDO (P);
END_STEP

ACTION ASetDO: #BEGIN_EDIT_BLOCK
do_LinkP1P2 := TRUE;

;#END_EDIT_BLOCK END_ACTION (*ASetDO*)
STEP S_Reset_DO:
AResetDO (P);
END_STEP

ACTION AResetDO: #BEGIN_EDIT_BLOCK
do_LinkP1P2 := FALSE;

;#END_EDIT_BLOCK END_ACTION (*AResetDO*)

(* transitions *)
TRANSITION Trans1 (* Trans1 *) FROM S_Init TO S_Idle :=  #BEGIN_EDIT_BLOCK
TRUE
;#END_EDIT_BLOCK
END_TRANSITION

GO_ON_TRANSITION TSetDO (* Trans2 *) FROM S_Idle TO S_Set_DO :=  #BEGIN_EDIT_BLOCK
bSetDO
;#END_EDIT_BLOCK
END_TRANSITION

GO_ON_TRANSITION TResetDO (* Trans3 *) FROM S_Set_DO TO S_Reset_DO :=  #BEGIN_EDIT_BLOCK
sv_PumpData[1].PumpState = nPumpStateFree OR
sv_PumpData[2].PumpState = nPumpStateFree
;#END_EDIT_BLOCK
END_TRANSITION

GO_ON_TRANSITION TIdle (* Trans4 *) FROM S_Reset_DO TO S_Idle :=  #BEGIN_EDIT_BLOCK
TRUE
;#END_EDIT_BLOCK
END_TRANSITION

(* end IecGraph-Code *)
(* sfc-code *)
(* end sfc-code *)

END_ALGORITHM

END_ALGORITHM_BLOCK

#END_OF_IEC_PART

@Puma @IecEditor 6 148 @Pou 25
@@@BEG_Comment@@@
@h    ! WARNING !
@h    The Kemro K2 system (including software) only meets category B according to EN 954-1,
@h    thus it is not intended for usage in safety-relevant control applications in the field
@h    of personal safety (e.g. emergency stop).
@h    To implement potentially necessary safety-relevant control tasks, always use additional
@h    external safety devices that are intended for the particular purpose, and meet the necessary
@h    functional safety.
@h    For further information see EN 954-1 (EN ISO 13849-1) and/or the K2-x00 user manual, chapter
@h    "CE conformity, directives and standards".

Algorithm block for setting hydraulic specific valves to link different pumps.
@@@END_Comment@@@

@BEG_Contents

@BEG_Func
@RT(17)FuncTreeContainer
0
@END_Func

@BEG_Const
@RT(18)ConstTreeContainer
0
@END_Const

@BEG_Export

@BEG_Kind
@ALGORITHM_BLOCK @RT(17)ABPumpCombination @STRUCTURED_TEXT
@RT(0) @RT(0) @RT(0)
@END_Kind

@BEG_Dcl
@RT(16)DclTreeContainer
4
@Var @RT(10)TaskInject @RT(0) @T @T @RENAMED 0 @T @T @DT @RT(4)TASK @RT(0) @T @T @BASIC 0 @F
@F @F
@T
@BEG_Attrib
3 @RT(0) @RT(0) @RT(0)
@END_Attrib
1 7 @F @F @F @F

@Var @RT(7)TaskMid @RT(0) @T @T @RENAMED 0 @T @T @DT @RT(4)TASK @RT(0) @T @T @BASIC 0 @F
@F @F
@T
@BEG_Attrib
3 @RT(0) @RT(0) @RT(0)
@END_Attrib
1 7 @F @F @F @F

@Var @RT(11)do_LinkP1P2 @RT(0) @T @F @DT @RT(4)BOOL @RT(0) @T @T @BASIC 0 @F
@F @F
@T
@BEG_Attrib
3 @RT(0) @RT(30)DO for linking Pump1 and Pump2 @RT(0)
@END_Attrib
1 8 @F @F @F @F

@Var @RT(11)sv_PumpData @RT(0) @T @T @DERIVED 0 @F @RT(10)tyPumpData @F
@T
@BEG_Attrib
3 @RT(0) @RT(0) @RT(0)
@END_Attrib
1 8 @F @F @F @F

@END_Dcl

@END_Export

@BEG_Body

2

@BEG_Export

@BEG_Algo
@PROCESS_ALGORITHM @RT(6)paInit @STRUCTURED_TEXT
@RT(0) @RT(0) @RT(7)TaskMid @T @F
@END_Algo

@BEG_Dcl
@RT(16)DclTreeContainer
0
@END_Dcl

@END_Export

@BEG_Export

@BEG_Algo
@PROCESS_ALGORITHM @RT(16)paLinkPump1Pump2 @SEQUENTIAL_FLOW_CHART
@RT(0) @RT(0) @RT(10)TaskInject @F @F
@END_Algo

@BEG_Dcl
@RT(16)DclTreeContainer
1
@Var @RT(6)bSetDO @RT(0) @T @T @RENAMED 0 @T @T @DT @RT(4)BOOL @RT(0) @T @T @BASIC 0 @F
@F @F
@T
@BEG_Attrib
3 @RT(0) @RT(0) @RT(0)
@END_Attrib
1 0 @F @F @F @F

@END_Dcl

@END_Export

@BEG_Body
@TL(12)
(**************************************** WARNING ********************************************
 *** The KEBA Kemro K2 System including software is not intended for safety control tasks! ***
 ***                       For further information see Comment tab!                        ***
 *********************************************************************************************)

IF IS_LINKED(do_LinkP1P2) THEN
   START_PROCESS_ALGORITHM(paLinkPump1Pump2);
END_IF;

STOP_PROCESS_ALGORITHM();

@END_Body

@@@BEG_Comment@@@
@TL(0)

@@@END_Comment@@@

@BEG_SfcBody
6 5 5

@BEG_SfcData 2
@StepSeq @RT(4)sseq @F 3
@Step @RT(6)S_Init @F @T @F @F @RT(0) @F
@AcbCont @RT(7)unnamed @F 0

@Trans @RT(6)Trans1 @F @T @F @F @T @T @TL(2)
TRUE

@RT(6)Trans1 @F
@Loop @RT(4)loop @F 2
@StepSeq @RT(3)seq @F 5
@Step @RT(6)S_Idle @F @F @F @F @RT(0) @F
@AcbCont @RT(7)unnamed @F 1
@Acb @RT(7)Action5 @F @T @RT(1)N @RT(0) @F @F @T @TL(5)
//set DO if a device actually outputs to both pumps
bSetDO := (sv_PumpData[1].PumpState = nPumpStateBusy) AND
          (sv_PumpData[2].PumpState = nPumpStateBusy) AND
          (sv_PumpData[1].ActiveDevice = sv_PumpData[2].ActiveDevice);

@F

@Trans @RT(6)TSetDO @F @T @F @F @T @F @TL(2)
bSetDO

@RT(6)Trans2 @F
@Step @RT(8)S_Set_DO @F @F @F @F @RT(0) @F
@AcbCont @RT(7)unnamed @F 1
@Acb @RT(6)ASetDO @F @T @RT(1)P @RT(0) @F @F @T @TL(2)
do_LinkP1P2 := TRUE;

@F

@Trans @RT(8)TResetDO @F @T @F @F @T @F @TL(3)
sv_PumpData[1].PumpState = nPumpStateFree OR
sv_PumpData[2].PumpState = nPumpStateFree

@RT(6)Trans3 @F
@Step @RT(10)S_Reset_DO @F @F @F @F @RT(0) @F
@AcbCont @RT(7)unnamed @F 1
@Acb @RT(8)AResetDO @F @T @RT(1)P @RT(0) @F @F @T @TL(2)
do_LinkP1P2 := FALSE;

@F

@Trans @RT(5)TIdle @F @T @T @T @T @F @TL(2)
TRUE

@RT(6)Trans4 @F

@END_SfcData
@SaActions 0
@SaTrans 0
@SaExits 0
@END_SfcBody

@@@BEG_Comment@@@
@TL(0)

@@@END_Comment@@@
@END_Body

@END_Contents

(* ---- ABPumpConnection.pu ---- *)
(*
@h    ! WARNING !
@h    The Kemro K2 system (including software) only meets category B according to EN 954-1,
@h    thus it is not intended for usage in safety-relevant control applications in the field
@h    of personal safety (e.g. emergency stop).
@h    To implement potentially necessary safety-relevant control tasks, always use additional
@h    external safety devices that are intended for the particular purpose, and meet the necessary
@h    functional safety.
@h    For further information see EN 954-1 (EN ISO 13849-1) and/or the K2-x00 user manual, chapter
@h    "CE conformity, directives and standards".
*)

IMPORT_OVER_LISTFILE
 CHECK_REF
, tyMovementRegisterList
, tsPumpConnectionList
, tyPumpConnectionList
, tsPumpConnectionElement

END_IMPORT

ALGORITHM_BLOCK ABPumpConnection #DUMMY_EDIT_BLOCK

SYSTEM_VAR
 sv_bInitDone : BOOL;
 sv_MovementsAvailable : tyMovementRegisterList;
 sv_iMovementsAvailable : DINT;
 sv_PumpConnectionList : tsPumpConnectionList;
END_VAR

SYSTEM_OBJECT
 TaskVis : TASK;
 PU_Task_7 : TASK;
END_OBJECT

POSTUPDATE_ALGORITHM pInitDone ON PU_Task_7 WITH sv_bInitDone

#BEGIN_EDIT_BLOCK
(**************************************** WARNING ********************************************
 *** The KEBA Kemro K2 System including software is not intended for safety control tasks! ***
 ***                       For further information see Comment tab!                        ***
 *********************************************************************************************)

START_PROCESS_ALGORITHM(paGetPumpConnectionVars);

;#END_EDIT_BLOCK END_ALGORITHM

PROCESS_ALGORITHM paGetPumpConnectionVars ON TaskVis

VAR_TEMP
 i : DINT;
 k : DINT;
END_VAR

VAR
 bFound : BOOL;
 tmpList : tyPumpConnectionList;
 tmpPumpConnection : tsPumpConnectionElement;
 bChanged : BOOL;
END_VAR
#BEGIN_EDIT_BLOCK
(**************************************** WARNING ********************************************
 *** The KEBA Kemro K2 System including software is not intended for safety control tasks! ***
 ***                       For further information see Comment tab!                        ***
 *********************************************************************************************)

//get references to "required pumps" variables and store them
//in a sv_PumpConnectionList
FOR i := 1 TO sv_iMovementsAvailable DO
   IF CHECK_REF(sv_MovementsAvailable[i].pMovementData^.AnaOutData.pRequiredPumps^) THEN
      //only add reference if it is not already in the list
      bFound := FALSE;
      FOR k := 1 TO sv_PumpConnectionList.iCount DO
         IF (sv_PumpConnectionList.Movements[k] = sv_MovementsAvailable[i].pMovementData^.AnaOutData.pRequiredPumps) THEN
            bFound := TRUE;
            EXIT;
         END_IF;
      END_FOR;

      IF NOT bFound THEN
         sv_PumpConnectionList.iCount := sv_PumpConnectionList.iCount + 1;
         sv_PumpConnectionList.Movements[sv_PumpConnectionList.iCount] := sv_MovementsAvailable[i].pMovementData^.AnaOutData.pRequiredPumps;
      END_IF;
   END_IF;
END_FOR;

//sort list depending on iOrder
//lowest number will be at the beginning of the list
tmpList := sv_PumpConnectionList.Movements;
bChanged := TRUE;
WHILE bChanged DO
   bChanged := FALSE;
   FOR i := 1 TO (sv_PumpConnectionList.iCount - 1) DO
      IF tmpList[(i+1)]^.iOrder < tmpList[i]^.iOrder THEN
         //change necessary
         tmpPumpConnection := tmpList[i];
         tmpList[i] := tmpList[i+1];
         tmpList[i+1] := tmpPumpConnection;
         bChanged := TRUE;
      END_IF;
   END_FOR;
END_WHILE;

//copy tmp list to SV
sv_PumpConnectionList.Movements := tmpList;

STOP_PROCESS_ALGORITHM();

;#END_EDIT_BLOCK END_ALGORITHM

END_ALGORITHM_BLOCK

#END_OF_IEC_PART

@Puma @IecEditor 6 148 @Pou 25
@@@BEG_Comment@@@
@h    ! WARNING !
@h    The Kemro K2 system (including software) only meets category B according to EN 954-1,
@h    thus it is not intended for usage in safety-relevant control applications in the field
@h    of personal safety (e.g. emergency stop).
@h    To implement potentially necessary safety-relevant control tasks, always use additional
@h    external safety devices that are intended for the particular purpose, and meet the necessary
@h    functional safety.
@h    For further information see EN 954-1 (EN ISO 13849-1) and/or the K2-x00 user manual, chapter
@h    "CE conformity, directives and standards".
@@@END_Comment@@@

@BEG_Contents

@BEG_Func
@RT(17)FuncTreeContainer
1
@Var @RT(9)CHECK_REF @RT(0) @T @T @DERIVED 0 @F @RT(23)KEBA_STANDARD_PROCEDURE @F
@T
@BEG_Attrib
0 @RT(0) @RT(0)
@END_Attrib
1 1 @F @F @F @F

@END_Func

@BEG_Const
@RT(18)ConstTreeContainer
0
@END_Const

@BEG_Export

@BEG_Kind
@ALGORITHM_BLOCK @RT(16)ABPumpConnection @STRUCTURED_TEXT
@RT(0) @RT(0) @RT(0)
@END_Kind

@BEG_Dcl
@RT(16)DclTreeContainer
6
@Var @RT(12)sv_bInitDone @RT(0) @T @T @RENAMED 0 @T @T @DT @RT(4)BOOL @RT(0) @T @T @BASIC 0 @F
@F @F
@T
@BEG_Attrib
3 @RT(0) @RT(0) @RT(0)
@END_Attrib
1 8 @F @F @F @F

@Var @RT(21)sv_MovementsAvailable @RT(0) @T @T @DERIVED 0 @F @RT(22)tyMovementRegisterList @F
@T
@BEG_Attrib
3 @RT(0) @RT(0) @RT(0)
@END_Attrib
1 8 @F @F @F @F

@Var @RT(22)sv_iMovementsAvailable @RT(0) @T @F @DT @RT(4)DINT @RT(0) @T @T @BASIC 0 @F
@F @F
@T
@BEG_Attrib
3 @RT(0) @RT(0) @RT(0)
@END_Attrib
1 8 @F @F @F @F

@Var @RT(21)sv_PumpConnectionList @RT(0) @T @T @DERIVED 0 @F @RT(20)tsPumpConnectionList @F
@T
@BEG_Attrib
3 @RT(0) @RT(0) @RT(0)
@END_Attrib
1 8 @F @F @F @F

@Var @RT(7)TaskVis @RT(0) @T @T @RENAMED 0 @T @T @DT @RT(4)TASK @RT(0) @T @T @BASIC 0 @F
@F @F
@T
@BEG_Attrib
3 @RT(0) @RT(0) @RT(0)
@END_Attrib
1 7 @F @F @F @F

@Var @RT(9)PU_Task_7 @RT(0) @T @T @RENAMED 0 @T @T @DT @RT(4)TASK @RT(0) @T @T @BASIC 0 @F
@F @F
@T
@BEG_Attrib
3 @RT(0) @RT(0) @RT(0)
@END_Attrib
1 7 @F @F @F @F

@END_Dcl

@END_Export

@BEG_Body

2

@BEG_Export

@BEG_Algo
@POSTUPDATE_ALGORITHM @RT(9)pInitDone @STRUCTURED_TEXT
@RT(0) @RT(12)sv_bInitDone @RT(9)PU_Task_7 @F @F
@END_Algo

@BEG_Dcl
@RT(16)DclTreeContainer
0
@END_Dcl

@END_Export

@BEG_Export

@BEG_Algo
@PROCESS_ALGORITHM @RT(23)paGetPumpConnectionVars @STRUCTURED_TEXT
@RT(0) @RT(0) @RT(7)TaskVis @F @F
@END_Algo

@BEG_Dcl
@RT(16)DclTreeContainer
6
@Var @RT(1)i @RT(0) @T @F @DT @RT(4)DINT @RT(0) @T @T @BASIC 0 @F
@F @F
@T
@BEG_Attrib
3 @RT(0) @RT(0) @RT(0)
@END_Attrib
1 4 @F @F @F @F

@Var @RT(1)k @RT(0) @T @F @DT @RT(4)DINT @RT(0) @T @T @BASIC 0 @F
@F @F
@T
@BEG_Attrib
3 @RT(0) @RT(0) @RT(0)
@END_Attrib
1 4 @F @F @F @F

@Var @RT(6)bFound @RT(0) @T @F @DT @RT(4)BOOL @RT(0) @T @T @BASIC 0 @F
@F @F
@T
@BEG_Attrib
3 @RT(0) @RT(0) @RT(0)
@END_Attrib
1 0 @F @F @F @F

@Var @RT(7)tmpList @RT(0) @T @T @DERIVED 0 @F @RT(20)tyPumpConnectionList @F
@T
@BEG_Attrib
3 @RT(0) @RT(0) @RT(0)
@END_Attrib
1 0 @F @F @F @F

@Var @RT(17)tmpPumpConnection @RT(0) @T @T @DERIVED 0 @F @RT(23)tsPumpConnectionElement @F
@T
@BEG_Attrib
3 @RT(0) @RT(0) @RT(0)
@END_Attrib
1 0 @F @F @F @F

@Var @RT(8)bChanged @RT(0) @T @F @DT @RT(4)BOOL @RT(0) @T @T @BASIC 0 @F
@F @F
@T
@BEG_Attrib
3 @RT(0) @RT(0) @RT(0)
@END_Attrib
1 0 @F @F @F @F

@END_Dcl

@END_Export

@BEG_Body
@TL(7)
(**************************************** WARNING ********************************************
 *** The KEBA Kemro K2 System including software is not intended for safety control tasks! ***
 ***                       For further information see Comment tab!                        ***
 *********************************************************************************************)

START_PROCESS_ALGORITHM(paGetPumpConnectionVars);

@END_Body

@@@BEG_Comment@@@
@TL(0)

@@@END_Comment@@@

@BEG_Body
@TL(47)
(**************************************** WARNING ********************************************
 *** The KEBA Kemro K2 System including software is not intended for safety control tasks! ***
 ***                       For further information see Comment tab!                        ***
 *********************************************************************************************)

//get references to "required pumps" variables and store them
//in a sv_PumpConnectionList
FOR i := 1 TO sv_iMovementsAvailable DO
   IF CHECK_REF(sv_MovementsAvailable[i].pMovementData^.AnaOutData.pRequiredPumps^) THEN
      //only add reference if it is not already in the list
      bFound := FALSE;
      FOR k := 1 TO sv_PumpConnectionList.iCount DO
         IF (sv_PumpConnectionList.Movements[k] = sv_MovementsAvailable[i].pMovementData^.AnaOutData.pRequiredPumps) THEN
            bFound := TRUE;
            EXIT;
         END_IF;
      END_FOR;

      IF NOT bFound THEN
         sv_PumpConnectionList.iCount := sv_PumpConnectionList.iCount + 1;
         sv_PumpConnectionList.Movements[sv_PumpConnectionList.iCount] := sv_MovementsAvailable[i].pMovementData^.AnaOutData.pRequiredPumps;
      END_IF;
   END_IF;
END_FOR;

//sort list depending on iOrder
//lowest number will be at the beginning of the list
tmpList := sv_PumpConnectionList.Movements;
bChanged := TRUE;
WHILE bChanged DO
   bChanged := FALSE;
   FOR i := 1 TO (sv_PumpConnectionList.iCount - 1) DO
      IF tmpList[(i+1)]^.iOrder < tmpList[i]^.iOrder THEN
         //change necessary
         tmpPumpConnection := tmpList[i];
         tmpList[i] := tmpList[i+1];
         tmpList[i+1] := tmpPumpConnection;
         bChanged := TRUE;
      END_IF;
   END_FOR;
END_WHILE;

//copy tmp list to SV
sv_PumpConnectionList.Movements := tmpList;

STOP_PROCESS_ALGORITHM();

@END_Body

@@@BEG_Comment@@@
@TL(0)

@@@END_Comment@@@
@END_Body

@END_Contents
